// TIA Portal V21 export
VAR_GLOBAL   // PLC tag table "ANALOG"
   "DOOR1 PRESSURE" AT %IW120 : Int;
   "DOOR2 PRESSURE" AT %IW122 : Int;
   "JACKET PRESSURE" AT %IW124 : Int;
   "CHAMBER PRESSURE" AT %IW126 : Int;
END_VAR
